Universal Robots PolyScope program: ur5e_force_Tcp_IP.urp

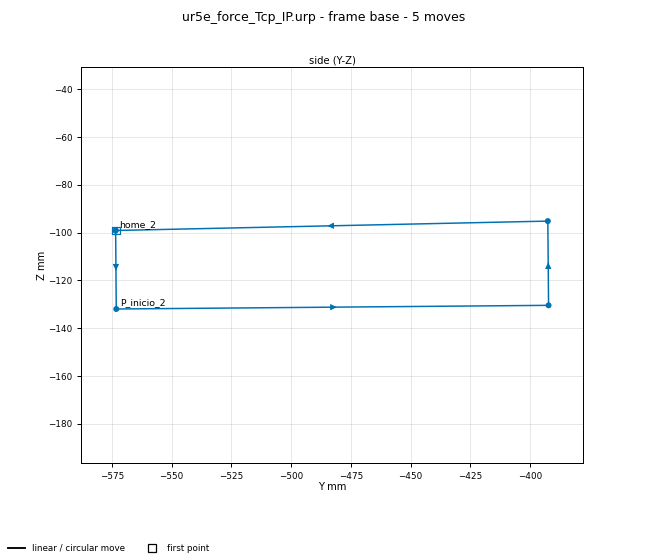
[picture p0: tool path of ur5e_force_Tcp_IP.urp in frame base, 5 of 5 moves have a stored position in this frame; points joined in program order, loops and branches not executed]
Program ur5e_force_Tcp_IP (installation=Testea_pruebas_spin directory=/programs/usbdisk createdIn=5.3.0.64176 lastSavedIn=5.3.0.64176 robotSerialNumber=20185500838)
Calibrated DH parameters: a=[0.000228, -0.232264, -0.085938, 0.000042, 0.000178, 0]; d=[0.162578, 124.608611, -334.653925, 210.179064, 0.099521, 0.099504]; alpha=[1.569639, -0.002858, 0.001822, 1.569892, -1.569434, 0]; deltaTheta=[0, -0.992947, 5.926272, 1.349872, 0.000001, 0]
Robot Program (runOnlyOnce=false)
  var_send := False
  fuerza := [0,0,30,0,0,0]
  vel := [0.1,0.1,0.1,0.17,0.17,0.17]
  vel_2 := [0.01,0.01,3,0.17,0.17,0.17]
  sel := [0,0,1,0,0,0]
  Incpos := [0.1,0,0,0,0,0]
  IncZ := [0,0,0.05,0,0,0]
  open := socket_open("192.168.0.10",5000)
  Script: socket_send_string("get")
  Script: textmsg("conexion establecida")
  Script: force_mode_set_damping(0.5)
  Script: force_mode_set_gain_scaling(1)
  SuppressedNode
    MoveL speed 250 mm/s, acceleration 1200 mm/s^2 (useActiveTCP=true) feature=Plano_mesa
      Wait Sleep waitTime=1
      Waypoint home: TCP in base x=247.306 y=-483.669 z=-99.139 mm, rx=-3.1347 ry=-0.0001 rz=-0.013 rad; joints [102.556, -47.246, 116.448, -158.848, -89.373, 192.746] deg; TCP offset x=0 y=0 z=107 mm, rx=0 ry=0 rz=0 rad; feature pose in base x=105.617 y=-391.736 z=-199.251 mm, rx=0.0085 ry=-0.0082 rz=0 rad
      var_send := True
      Script: zero_ftsensor()
      Wait Sleep waitTime=0.2
      Waypoint P_inicio_2: motionParameters(jointSpeed=1.047198 jointAcceleration=1.396263 cartesianSpeed=0.25 cartesianAcceleration=1.2); TCP in base x=344.87 y=-573.134 z=-131.926 mm, rx=-3.1347 ry=-0.0001 rz=-0.013 rad; joints [109.236, -35.121, 92.965, -147.556, -89.384, 199.412] deg; TCP offset x=0 y=0 z=107 mm, rx=0 ry=0 rz=0 rad; feature pose in base x=105.617 y=-391.736 z=-199.251 mm, rx=0.0085 ry=-0.0082 rz=0 rad
      P_iniciodef := get_actual_tcp_pose()
      Script: force_mode(Joint_6_name,sel,fuerza,2,vel)
      Wait Sleep waitTime=2
      SuppressedNode
        P_final := pose_add(P_iniciodef, Incpos)
      SuppressedNode
        Waypoint Waypoint (Variable): motionParameters(jointSpeed=1.047198 jointAcceleration=1.396263 cartesianSpeed=0.05 cartesianAcceleration=1.2); variable=P_final
      Waypoint P_finaldef_2: motionParameters(jointSpeed=1.047198 jointAcceleration=1.396263 cartesianSpeed=0.05 cartesianAcceleration=1.2); TCP in base x=344.863 y=-392.309 z=-130.394 mm, rx=-3.1347 ry=-0.0001 rz=-0.013 rad; joints [116.176, -43.693, 119.171, -165.262, -89.332, 206.379] deg; TCP offset x=0 y=0 z=107 mm, rx=0 ry=0 rz=0 rad
      Script: end_force_mode()
      Wait Sleep waitTime=0.5
      SuppressedNode
        P_final_salida := pose_add(P_finaldef_2, IncZ)
      Waypoint P_salida_2: TCP in base x=344.584 y=-392.616 z=-95.16 mm, rx=-3.1347 ry=-0.0001 rz=-0.0131 rad; joints [116.141, -48.931, 120.117, -160.971, -89.316, 206.332] deg
      Waypoint home: TCP in base x=247.306 y=-483.669 z=-99.139 mm, rx=-3.1347 ry=-0.0001 rz=-0.013 rad; joints [102.556, -47.246, 116.448, -158.848, -89.373, 192.746] deg; feature pose in base x=105.617 y=-391.736 z=-199.251 mm, rx=0.0085 ry=-0.0082 rz=0 rad
      var_send := False
      Halt
  MoveL speed 250 mm/s, acceleration 1200 mm/s^2 (useActiveTCP=true) feature=Plano_mesa
    Wait Sleep waitTime=1
    Waypoint home_2: TCP in base x=344.626 y=-573.395 z=-99.088 mm, rx=-3.1348 ry=-0.0001 rz=-0.0131 rad; joints [109.213, -38.808, 93.748, -144.653, -89.374, 199.383] deg; feature pose in base x=105.617 y=-391.736 z=-199.251 mm, rx=0.0085 ry=-0.0082 rz=0 rad
    var_send := True
    Script: zero_ftsensor()
    Wait Sleep waitTime=0.2
    Waypoint P_inicio_2: TCP in base x=344.87 y=-573.134 z=-131.926 mm, rx=-3.1347 ry=-0.0001 rz=-0.013 rad; joints [109.236, -35.121, 92.965, -147.556, -89.384, 199.412] deg; TCP offset x=0 y=0 z=107 mm, rx=0 ry=0 rz=0 rad
    SuppressedNode
      P_iniciodef := get_actual_tcp_pose()
    Script: force_mode(Joint_6_name,sel,fuerza,2,vel)
    Wait Sleep waitTime=2
    SuppressedNode
      P_final := pose_add(P_iniciodef, Incpos)
    SuppressedNode
      Waypoint Waypoint (Variable): motionParameters(jointSpeed=1.047198 jointAcceleration=1.396263 cartesianSpeed=0.05 cartesianAcceleration=1.2); variable=P_final
    Waypoint P_finaldef_2: motionParameters(jointSpeed=1.047198 jointAcceleration=1.396263 cartesianSpeed=0.05 cartesianAcceleration=1.2); TCP in base x=344.863 y=-392.309 z=-130.394 mm, rx=-3.1347 ry=-0.0001 rz=-0.013 rad; joints [116.176, -43.693, 119.171, -165.262, -89.332, 206.379] deg; TCP offset x=0 y=0 z=107 mm, rx=0 ry=0 rz=0 rad
    Script: end_force_mode()
    Wait Sleep waitTime=0.5
    SuppressedNode
      P_final_salida := pose_add(P_finaldef_2, IncZ)
    Waypoint P_salida_2: TCP in base x=344.584 y=-392.616 z=-95.16 mm, rx=-3.1347 ry=-0.0001 rz=-0.0131 rad; joints [116.141, -48.931, 120.117, -160.971, -89.316, 206.332] deg
    SuppressedNode
      Waypoint home: TCP in base x=247.306 y=-483.669 z=-99.139 mm, rx=-3.1347 ry=-0.0001 rz=-0.013 rad; joints [102.556, -47.246, 116.448, -158.848, -89.373, 192.746] deg; feature pose in base x=105.617 y=-391.736 z=-199.251 mm, rx=0.0085 ry=-0.0082 rz=0 rad
    Waypoint home_2: motionParameters(jointSpeed=1.047198 jointAcceleration=1.396263 cartesianSpeed=0.25 cartesianAcceleration=1.2); TCP in base x=344.626 y=-573.395 z=-99.088 mm, rx=-3.1348 ry=-0.0001 rz=-0.0131 rad; joints [109.213, -38.808, 93.748, -144.653, -89.374, 199.383] deg; feature pose in base x=105.617 y=-391.736 z=-199.251 mm, rx=0.0085 ry=-0.0082 rz=0 rad
    var_send := False
    Halt
Thread Thread_1 (runOnlyOnce=false trackProgramExecution=false)
  var_2 := force()
  var_1 := get_tcp_force()
  var_3 := norm(get_target_tcp_speed())
  var_4 := get_steptime()
  SuppressedNode
    Wait Sleep waitTime=0.1
  If var_send≟ True
    Script: socket_send_string(var_1)
    Script: socket_send_string(var_2)
    Script: socket_send_string("]")
    Script: socket_send_string(var_3)
    SuppressedNode
      Script: socket_send_string("]")
    SuppressedNode
      Script: socket_send_string(var_4)
  Else 
    SuppressedNode
      Script: socket_send_string("a")
  SuppressedNode
    Script: socket_send_string(var_1)
  SuppressedNode
    Script: socket_send_string("a")
  Script: sync()
